TYPE ST_MotionlinxAI_Axis_Config :
	STRUCT
		ExtendTime	: LREAL;
		RetractTime : LREAL;
	END_STRUCT
END_TYPE

(* stored: Version 1.1.0.1, ProductVersion 3.1.4024.15
   DUT ST_MotionlinxAI_Axis_Config: Id {f16f9533-2248-4a33-bc1e-96f6c88dabba} *)
